{attribute 'GeneratedUsingTerminal: EPP1322-0001-0017'}
{attribute addProperty BoxType "EPP1322-0001-0017"}
{attribute addProperty Id "RC20_AB1_EPP1008_0001EPP1008_78E8D3DD12RC20_AB2_EPP1008_0001EPP1008_78E8D3DD12RC20_AB6_EPP1008_0001EPP1008_78E8D3DD12RC20_AB3_EPP1008_0001EPP1008_78E8D3DD12RC20_AB4_EPP1008_0001EPP1008_78E8D3DD12RC20_AB7_EPP1008_0001EPP1008_78E8D3DD12RC20_AB9_EPP1008_0001EPP1008_78E8D3DD12RC20_AB10_EPP1008_0001EPP1008_78E8D3DD12RC20_AB8_EPP1008_0001EPP1008_78E8D3DD12RC20_AB5_EPP1008_0001EPP1008_78E8D3DD12"}
{attribute addProperty CRC "1507086522"}
{attribute addProperty Size "120"}
{attribute addProperty Name "RC20_EPP (EPP1322-0001)"}
TYPE RC20_EPP_EPP1322_0001_59D450BA EXTENDS EPP1322_1FC0878B :
STRUCT
	{attribute addProperty Name "RC20_AB1 (EPP1008-0001)"}
	{attribute addProperty PreviousPort "RC20_EPP (EPP1322-0001) : D"}
	RC20_AB1_EPP1008_0001 : EPP1008_78E8D3DD;
	{attribute addProperty Name "RC20_AB2 (EPP1008-0001)"}
	{attribute addProperty PreviousPort "RC20_AB1 (EPP1008-0001) : B"}
	RC20_AB2_EPP1008_0001 : EPP1008_78E8D3DD;
	{attribute addProperty Name "RC20_AB6 (EPP1008-0001)"}
	{attribute addProperty PreviousPort "RC20_AB2 (EPP1008-0001) : B"}
	RC20_AB6_EPP1008_0001 : EPP1008_78E8D3DD;
	{attribute addProperty Name "RC20_AB3 (EPP1008-0001)"}
	{attribute addProperty PreviousPort "RC20_AB6 (EPP1008-0001) : B"}
	RC20_AB3_EPP1008_0001 : EPP1008_78E8D3DD;
	{attribute addProperty Name "RC20_AB4 (EPP1008-0001)"}
	{attribute addProperty PreviousPort "RC20_AB3 (EPP1008-0001) : B"}
	RC20_AB4_EPP1008_0001 : EPP1008_78E8D3DD;
	{attribute addProperty Name "RC20_AB7 (EPP1008-0001)"}
	{attribute addProperty PreviousPort "RC20_EPP (EPP1322-0001) : B"}
	RC20_AB7_EPP1008_0001 : EPP1008_78E8D3DD;
	{attribute addProperty Name "RC20_AB9 (EPP1008-0001)"}
	{attribute addProperty PreviousPort "RC20_AB7 (EPP1008-0001) : B"}
	RC20_AB9_EPP1008_0001 : EPP1008_78E8D3DD;
	{attribute addProperty Name "RC20_AB10 (EPP1008-0001)"}
	{attribute addProperty PreviousPort "RC20_AB9 (EPP1008-0001) : B"}
	RC20_AB10_EPP1008_0001 : EPP1008_78E8D3DD;
	{attribute addProperty Name "RC20_AB8 (EPP1008-0001)"}
	{attribute addProperty PreviousPort "RC20_AB10 (EPP1008-0001) : B"}
	RC20_AB8_EPP1008_0001 : EPP1008_78E8D3DD;
	{attribute addProperty Name "RC20_AB5 (EPP1008-0001)"}
	{attribute addProperty PreviousPort "RC20_AB8 (EPP1008-0001) : B"}
	RC20_AB5_EPP1008_0001 : EPP1008_78E8D3DD;
END_STRUCT
END_TYPE

(* stored: Version 1.2.0.0, ProductVersion 3.1.4024.11
   DUT RC20_EPP_EPP1322_0001_59D450BA: Id {a999b69f-f99e-0153-1229-7c6b29e73577} *)
